	bSetParameter					: BOOL;
	bConnect						: BOOL := TRUE;
	bIncommingMsg					: BOOL;
	hrErrorOccurred 				: DINT; //Contains latest error message
	sTopicRec						: STRING(255);
	sMessage						: STRING(255);
	ReinitComParams					: BOOL;
	
	
	bSubscribed						: BOOL;
	ton_PublishInterval				: TON;
	sPubTopic						: STRING;
	sSubTopic						: STRING;
	
	stPubDataMaster					: ST_InterMachineCom_Master;
	stPubDataSlave					: st_InterMachineCom_Slave;
	stSubDataMaster					: ST_InterMachineCom_Master;
	stSubDataSlave					: st_InterMachineCom_Slave;
	
	
	fbJson         	: FB_JsonSaxWriter;
  	fbJsonDataType 	: FB_JsonReadWriteDataType;
	sJsonDocPub     : STRING(255);
	bRecJsonOK		: BOOL;
	
	
	sMasterTopic 	: STRING := 'master';
END_VAR

(* 
Internal broker is used to post local data in the master topic. The unit listens to the slave topics

*)

//Connect brokers

//Generate machinedata for internal master
InternalBroker(bConnect := TRUE, sHostname := ST_params.InternalBrokerIP);
InternalBroker.Publish(
	Interval := st_params.MasterPublishRate, 
	sTopic := sMasterTopic, 
	sMessage := StructToJson(TRUE));
InternalBroker.Subscribe(sTopic := 'slave/epu/#/read');

IF internalbroker.bIncomingMsg THEN
	JsonToStruct(sMessage := internalbroker.sMessage);
END_IF

//Generate slave data for the external master
ExternalBroker(bConnect := SlaveConnectionData.enable, sHostname := SlaveConnectionData.BrokerIP);
ExternalBroker.Publish(Interval := st_params.SlavePublishRate, 
		sTopic := CONCAT(CONCAT('epu/slave/',settings.Properties.s_SerialNumber),'/read'),
		sMessage := StructToJson(FALSE));
ExternalBroker.Subscribe(sTopic := sMasterTopic);

IF Externalbroker.bIncomingMsg THEN
	JsonToStruct();
END_IF




//Publish as master 
sPubTopic := 'master';
sSubTopic := 'slave/#';
//Ton_PublishInterval.PT := st_params.MasterPublishRate;
//generate json doc
fbJson.ResetDocument();
fbJsonDataType.AddJsonValueFromSymbol(fbJson, 'ST_InterMachineCom_Master', SIZEOF(stPubDataMaster), ADR(stPubDataMaster));
fbJson.EndObject();
fbJson.CopyDocument(sJsonDocPub, SIZEOF(sJsonDocPub));

IF SlaveConnectionData.enable AND SlaveConnectionData.BrokerIP <> '' THEN
	sSubTopic := 'master';
	sPubTopic := CONCAT('slave/', settings.Properties.s_SerialNumber);
	Ton_PublishInterval.PT := st_params.MasterPublishRate;
	//generate json doc
	fbJson.ResetDocument();
	fbJsonDataType.AddJsonValueFromSymbol(fbJson, 'ST_InterMachineCom_Slave', SIZEOF(stPubDataSlave), ADR(stPubDataSlave));
	fbJson.EndObject();
	fbJson.CopyDocument(sJsonDocPub, SIZEOF(sJsonDocPub));
	
	//converter receiving message back to structur
	fbJsonDataType.SetSymbolFromJson(sMessage, 'st_InterMachineCom_Master', SIZEOF(stSubDataMaster), ADR(stSubDataMaster));
END_IF

// publish
IF fbMqttClientInternal.bConnected THEN
    IF NOT bSubscribed THEN
        bSubscribed := fbMqttClientInternal.Subscribe(sTopic:=sSubTopic, eQoS:=TcIotMqttQos.AtMostOnceDelivery); //sSubTopic
    END_IF
    ton_PublishInterval(IN:=TRUE);
    IF ton_PublishInterval.Q THEN // publish new payload every second
        ton_PublishInterval(IN:=FALSE);
			fbMqttClientInternal.Publish(sTopic:=sPubTopic,
			pPayload := ADR(sJsonDocPub),
			nPayloadSize := LEN2(ADR(sJsonDocPub)),
			eQoS := TcIotMqttQos.AtMostOnceDelivery,
			bRetain:= TRUE,
			bQueue := FALSE);
    END_IF
END_IF


IF bIncommingMsg THEN
	bRecJsonOK := fbJsonDataType.SetSymbolFromJson(sMessage, 'st_InterMachineCom_Slave', SIZEOF(stSubDataSlave), ADR(stSubDataSlave));
END_IF

Internalbroker.Subscribe();

METHOD CheckSlaves : BOOL
VAR_INPUT
END_VAR
END_METHOD

METHOD GetSubData : BOOL
VAR_INPUT
END_VAR
END_METHOD

METHOD JsonToStruct : BOOL
VAR_INPUT
	MasterMode		: BOOL;
END_VAR

VAR_IN_OUT
	sMessage : STRING;
END_VAR
IF MasterMode THEN
	//Get the message from the external broker 'master' subscribtion, format according to ST_IntermachineCom_Master
ELSE
	//Get the message from the internal broker '+/slave/#/read' subscriptiom, format according to ST_intermachineCom_Slave
	(* A json parser need to be constructed such that the combined json struct is formatted in separate st_IntermachineCom_slave structs.
	
	Data can come from the epu or hpu and distinquish is made through the topic path: /slave/hpu/#, or /slave/epu/#
	For example the epu slave path is: /slave/epu/{serialnumber}/read and the ST_intermachineCom_slave struct comes out.
	A json filter has to be made to iterate along all serial numbers in epu and hpu group. 
	A method must be created where the data is temporarily stored such that the ACP (available charge power), 
	ADP (available discharge power) and ARP (available reactive power) can me summed and used for the power setpoint calculation.
	
	A separate topic /slave/epu/{serialnumber}/write can be used to control slaves individually with the ST_IntermachineCom_master struct.
	However, this requires the slave CW heartbeat and SW heartbeat to be updated within heartbeat time limit. When the CW heartbeat stops, 
	the slave will go to general operation related to the 'master' topic that is broadcasted. 
	*)
END_IF
END_METHOD

METHOD Reset : BOOL
VAR_INPUT
END_VAR
IF InternalBroker.bRestartConnection AND ExternalBroker.bRestartConnection THEN
	InternalBroker.bRestartConnection := FALSE;
	ExternalBroker.bRestartConnection := FALSE;
	Reset := TRUE;
ELSE
	InternalBroker.bRestartConnection := NOT InternalBroker.bRestartConnection;
	ExternalBroker.bRestartConnection := NOT ExternalBroker.bRestartConnection;
END_IF
END_METHOD

METHOD SetPubData : BOOL
VAR_INPUT
END_VAR

VAR_INST
	WatchdogPulse	: TON; 
END_VAR
WatchdogPulse(IN := NOT watchdogPulse.Q, PT:= st_params.WatchdogPulseRate);

//Internal 'master' data to control slaves
stPubDataMaster.CW.0 := monitor.powerstack.b_StartedState;
stPubDataMaster.CW.1 := monitor.powerstack.e_State = eStatusPowerstack.idle;
stPubDataMaster.CW.2 := monitor.powerstack.e_State = eStatusPowerstack.shutdown;
stPubDataMaster.CW.3 := GVL.b_EmergencyShutdownActive AND ST_IntermachineCom_params.EMstopCoupling;
stPubDataMaster.CW.4 := monitor.system.e_State = eSystemState.Reset;
stPubDataMaster.CW.15 := SEL(watchdogPulse.Q, stPubDataMaster.CW.15, NOT stPubDataMaster.CW.15);
stPubDataMaster.PS := 0; // TBD based on slaves
stPubDataMaster.QS := 0; 

//Slave data for external master
stPubDataSlave.ACP := TO_UINT(ABS(monitor.powerstack.r_Pmin));
stPubDataSlave.ADP := TO_UINT(ABS(monitor.powerstack.r_PMax));
stPubDataSlave.AQ := TO_UINT(ABS(monitor.powerstack.r_QMax));
stPubDataSlave.SW.0 := monitor.system.e_State = eSystemState.StandBy OR monitor.system.e_State = eSystemState.Conditioning;
stPubDataSlave.SW.1 := monitor.powerstack.b_StartedState;
stPubDataSlave.SW.2 := monitor.system.e_State = eSystemState.Stopped;
stPubDataSlave.SW.3 := monitor.system.e_State = eSystemState.Discharging_Only;
stPubDataSlave.SW.4 := monitor.system.e_State = eSystemState.Charging_Only;
stPubDataSlave.SW.5 := GVL.b_WarningActive;
stPubDataSlave.SW.6 := GVL.b_NormalShutdownActive;
stPubDataSlave.SW.7 := GVL.b_EmergencyShutdownActive;
stPubDataSlave.SW.15 := stSubDataMaster.CW.15;
END_METHOD

METHOD StructToJson : STRING
VAR_INPUT
	Mastermode		: BOOL; //if false, then slave mode
END_VAR
fbJson.ResetDocument();

IF MasterMode THEN
	fbJsonDataType.AddJsonValueFromSymbol(fbJson, 'ST_InterMachineCom_Master', SIZEOF(stPubDataMaster), ADR(stPubDataMaster));
ELSE
	fbJsonDataType.AddJsonValueFromSymbol(fbJson, 'ST_InterMachineCom_Slave', SIZEOF(stPubDataSlave), ADR(stPubDataSlave));
END_IF

fbJson.EndObject();
fbJson.CopyDocument(StructToJson, SIZEOF(StructToJson));
END_METHOD

END_FUNCTION_BLOCK

// ---- POUs/Objects/PLCStatus/FB_PLCUpdate.TcPOU
FUNCTION_BLOCK FB_PLCUpdate

VAR_INPUT
	bUpdate				: BOOL;
	bAbortUpdate		: BOOL;
END_VAR

VAR_OUTPUT
	FTPState			: eFTPstate;
	InstalState			: eInstalState;
	BackupState			: eInstalState;
	sLogMessage 		: STRING(255);
	bCheckUpdates		: BOOL;	
	bUpdateAvailable 	: BOOL;
END_VAR

VAR	
	rTrig_CheckUpdate	: R_Trig;
	
    fbFileDelete 		: FB_FileDelete;  (* Om oude bestanden te verwijderen *)
    
    sJsonUrl      		: STRING := 'http://server.com/updates.json'; (* JSON met update-info *)
    sUpdateUrl    		: STRING := '';  (* URL van het updatebestand uit JSON *)
    sLocalPath    		: STRING := '/usr/local/updates/update.tsmpkg';
    sBackupPath   		: STRING := '/usr/local/backup/old_version.tsmpkg';
    
    sCurrentVersion 	: STRING := '1.2.0';  (* Huidige versie van de PLC *)
    sNewVersion     	: STRING := '';       (* Nieuwe versie uit JSON *)

   
    bDownloadComplete 	: BOOL;
    bInstallComplete 	: BOOL;
    bRollbackNeeded 	: BOOL;
    eState 				: INT := 0;
    iRetryCount 		: INT := 0;
END_VAR




CASE eState OF
    0: // Controleer op update via JSON
		rTrig_CheckUpdate(CLK := bUpdate);
		IF rTrig_CheckUpdate THEN
			bCheckUpdates := TRUE;
		END_IF
		
		IF 
		CheckForUpdates();
        

    1: // Maak een backup van de huidige versie
		BackupState := Copy(sSrcPath := sLocalPath, sDestPath := sBackupPath);
		
        IF BackupState = eInstalState.Success THEN
            eState := 2;
		ELSIF BackupState = eInstalState.Failure OR bAbortUpdate THEN
			eState := 99;
        END_IF

    2: // Download de nieuwe update via FTP
		FTPState := DownloadUpdate(
			sHost := 'temp',
			sUsername := 'tempuser',
			sPassword := 'tempPass',
			sSrcFile := 'path/1',
			sDesFile := 'path/2',
			start :=  bUpdateAvailable);

        IF FTPState = eFTPState.Success THEN
            bDownloadComplete := TRUE;
            eState := 3;
        ELSIF FTPState = eFTPState.Failure OR bAbortUpdate THEN
                eState := 99; // Ga naar fallback
        END_IF

    3: // Wachten op bevestiging van de gebruiker via HMI
        IF bUpdate THEN
			bUpdateStarted := TRUE;
            eState := 4;
        END_IF

    4: // Installeer de update
		InstalState := Copy(sSrcPath := sLocalPath, sDestPath := 'path/2');
		IF InstalState = eInstalState.Success THEN
			bInstallComplete := TRUE;
			eState := 5;
		ELSIF InstalState = eInstalState.Failure OR bAbortUpdate THEN
			bRollbackNeeded := TRUE;
            eState := 6; // Ga naar rollback
		END_IF

    5: // Herstart de PLC na succesvolle update
        SystemReboot();

    6: // Rollback uitvoeren als de update is mislukt
		InstalState := Copy(sSrcPath := sBackupPath,  sDestPath := '/usr/local/boot/update.tsmpkg');

		IF InstalState = eInstalState.Success THEN
			SystemReboot();  // Herstart de PLC met oude versie
		ELSIF InstalState = eInstalState.Failure OR bAbortUpdate THEN
			eState := 99;  // Fallback activeren als rollback mislukt
		END_IF

    99: // Fallback: Stop het updateproces en meld de fout
        bUpdateAvailable := FALSE;
		bUpdateStarted := FALSE;
        bRollbackNeeded := FALSE;
        iRetryCount := 0;
END_CASE

CASE eState OF
    0:	sLogMessage := 'Check if update is available';
        WriteLog(sLogMessage);
        
   1:	sLogMessage := 'Create backup of current software';
        WriteLog(sLogMessage);

    2:	sLogMessage := 'Downloading update';
        WriteLog(sLogMessage);
		
	3:	sLogMessage := 'Update ready for installation';
		WriteLog(sLogMessage);
		
	4:	sLogMessage := 'Installing update';
		WriteLog(sLogMessage);
		
	5:	sLogMessage := 'Rebooting system';
		WriteLog(sLogMessage);    
		
    6:	sLogMessage := 'Update failed, rollback started';
         WriteLog(sLogMessage);
		 
    99:
        sLogMessage := 'Update mislukt, fallback geactiveerd';
        WriteLog(sLogMessage);
END_CASE

METHOD CheckForUpdates : BOOL
VAR_INPUT
	sServerUrl   : STRING := 'http://server.com/updates.json'; (* Volledige URL *)
END_VAR

VAR_INST
	fbHttpClient 		: FB_IotHttpClient;  (* Voor JSON versiecontrole *)
	     
    sResponse    : STRING(1024);  (* Buffer voor de server response *)
    bExecute     : BOOL := TRUE;
    bDone        : BOOL;
    bError       : BOOL;
END_VAR
fbHttpClient(
	sHostName := sHostName,
	


fbHttpClient.sHost := 'server.com';  // Vervang met je eigen server
fbHttpClient.sResource := '/updates.json';  // JSON-bestand
fbHttpClient.eMethod := E_HttpMethod.GET;
fbHttpClient.bExecute := TRUE;

IF fbHttpClient.eState = E_HttpRequestState.Done THEN
	sNewVersion := ExtractJsonValue(fbHttpClient.sResponseContent, 'latest_version');
	sUpdateUrl := ExtractJsonValue(fbHttpClient.sResponseContent, 'update_file');
	
	IF sNewVersion > sCurrentVersion THEN
		bUpdateAvailable := TRUE;
		eState := 1;
	END_IF
END_IF


(* Stap 1: HTTP Request starten *)
IF bExecute THEN
    fbHttpClient. := sServerUrl;   (* Geef de volledige URL mee *)
    fbHttpClient.eMethod := T_IotHttpMethod.Get;  (* HTTP GET Methode *)
    fbHttpClient.bExecute := TRUE;
    bExecute := FALSE; (* Voorkomt dat het telkens opnieuw start *)
END_IF

(* Stap 2: Wachten op antwoord *)
IF fbHttpClient.bDone THEN
    sResponse := fbHttpClient.sResponse;  (* Server response opslaan *)
    bDone := TRUE;
ELSIF fbHttpClient.bError THEN
    bError := TRUE;
END_IF
END_METHOD

METHOD Copy : eInstalstate
VAR_INPUT
	sSrcPath : STRING;
	sDestPath: STRING;
END_VAR

VAR_OUTPUT
	Busy 		: BOOL;
    Error 		: BOOL;
	ErrID 		: UDINT;
END_VAR

VAR_INST
	ton_waitRetry		: ton := (pt := T#2S);
	fbFileCopy   		: FB_FileCopy;    (* Voor het maken van een backup *)
END_VAR
fbFileCopy(
	sSrcPathName := sSrcPath,
	sDestPathName := sDestPath,
	tTimeOut := T#15S,
	bBusy => Busy,
	bError => Error,
	nErrId => ErrID);
	
ton_waitRetry(Q => fbFileCopy.bExecute);

IF Error THEN
	Copy := eInstalState.Failure;
ELSIF busy THEN
	Copy := eInstalState.InProgress;
	ton_waitRetry.IN := FALSE;
ELSE
	IF NOT fbFileCopy.bExecute THEN
		Copy := eInstalState.Success;
	END_IF
	ton_waitRetry.IN := TRUE;
END_IF
END_METHOD

METHOD DownloadUpdate : eFTPState

VAR_INPUT
	sHost 			: STRING := 'ftp.example.com';
	sUsername		: STRING;
	sSrcFile		: STRING;
	sDesFile		: STRING;
	sPassword		: STRING;
	Start			: BOOL;
END_VAR

VAR_OUTPUT
	Busy 		: BOOL;
    Error 		: BOOL;
	ErrID 		: UDINT;
END_VAR

VAR_INST
	bRetry			: BOOL;
	byMaxRetries	: BYTE := 3;
	byRetryCounter	: BYTE;
	StartTrigger : R_TRIG;	
	FTPstate 	: eFTPState;
	ftpOpen 	: FB_FTP_Open; 			// Function block om verbinding te openen.
	ftpDownload : FB_FTP_FileDownload; 	// Function block om het bestand te downloaden
    ftpClose 	: FB_FTP_Close;  			// Function block om de verbinding te sluiten
    hFTP 		: T_HFTP; //FTP handle / identifyer
	RTrig_Error	: R_Trig;
END_VAR
StartTrigger(CLK:= start);

CASE FTPState OF
      eFTPState.Disconnected:
			IF StartTrigger.Q OR bRetry THEN
				bRetry := FALSE;
      			FTPState := eFTPState.Connecting;
			END_IF
			
     eFTPState.Connecting:
         ftpOpen(
			sHost:= sHost,
			nPort:= 21,
			sUsername:= sUsername,
			sPassword:= sPassword,
			tTimeout:= T#15S,
			bExecute := TRUE,
			hFTP=> hFTP,
			bBusy => busy,
			bError => Error,
			nErrID=> ErrID
			);
         IF NOT Busy AND NOT Error THEN
             ftpOpen(bExecute:= FALSE);
             FTPState := eFTPstate.Downloading;
         END_IF
		 
     eFTPstate.Downloading:
		ftpDownload(
			sNetID:= '',              // Lokale machine
			hFTP:= hFTP,              // Gebruik de handle van de geopende verbinding
			sSrcFile:= '\TestFolder\File1.txt',
            sDesFile:= '\Program Files\TestFile1.txt',
			tTimeout:= T#15S,         // Timeout
			bexecute := TRUE,
			bBusy => busy,
            bError => error,
			nErrID=> ErrID
		);
         IF NOT busy AND NOT Error THEN
             ftpDownload(bExecute:= FALSE);
             FTPState := eFTPState.Success;
         END_IF
     eFTPState.Success:
		ftpClose(
			sNetID:= '',              // Lokale machine
			hFTP:= hFTP,              // Gebruik de handle van de geopende verbinding
			bExecute:= TRUE,      // Start het sluiten van de verbinding
			bBusy => busy,
            bError => error,
			tTimeout:= T#15S,         // Timeout
			nErrID=> ErrID
		);
	 	
       	 IF NOT busy AND NOT Error THEN
             ftpClose(bExecute:= FALSE);
             FTPstate := eFTPState.Disconnected;
			 byRetryCounter := 0;
         END_IF
		
	eFTPState.Failure:
		IF StartTrigger.Q THEN
			FTPState := eFTPState.Connecting;
		END_IF	 	
END_CASE

//Retry on error trigger
RTrig_Error(CLK:= Error);
IF RTrig_Error.Q THEN
	IF ByRetryCounter < byMaxRetries THEN
		FTPstate := eFTPState.Disconnected;
		bRetry := TRUE;
		byRetryCounter := byRetryCounter +1;
	ELSE
		FTPstate := eFTPState.Failure;
	END_IF
END_IF

DownloadUpdate := FTPState;
END_METHOD

METHOD SystemReboot : BOOL
VAR_INPUT
END_VAR

VAR_INST
    fbSysRestart 		: TC_Restart; (* Systeemherstartfunctie *)
END_VAR
fbSysRestart();
END_METHOD

METHOD WriteLog : BOOL
VAR_INPUT
    sMessage : STRING;
END_VAR

VAR_INST
    fbLogWriter 		: FB_FileWrite;
END_VAR
fbLogWriter(
fbLogWriter.sFileName := '/usr/local/logs/update_log.txt';
fbLogWriter.sData := sMessage + Char(13) + Char(10);
fbLogWriter.bExecute := TRUE;
WriteLog := fbLogWriter.bDone;
END_METHOD

END_FUNCTION_BLOCK

// ---- POUs/System/PowerControl/fb_measurementCheck.TcPOU
FUNCTION_BLOCK fb_measurementCheck
VAR_IN_OUT
	r_in : REAL;
END_VAR
VAR_INPUT
	b_externalFault : BOOL;
	r_LowLimit	 	: REAL;
	r_HighLimit		: REAL;
	by_Mode			: BYTE := 0; // 0= min, 1= avg, 2= Max, 3=SUM
END_VAR

VAR
	by_InputOK		: BYTE;
END_VAR

VAR_OUTPUT
	r_Out			: REAL;
	Q				: BOOL;
END_VAR


//Check if values are within set ranges
by_InputOK.0 := r_in > r_LowLimit AND r_in < r_HighLimit;
by_InputOK.1 := r_in[Phases.L1] > r_LowLimit AND r_in[phases.L1] < r_HighLimit;
by_InputOK.2 := r_in[Phases.L2] > r_LowLimit AND r_in[phases.L2] < r_HighLimit;
by_InputOK.3 := r_in[Phases.L3] > r_LowLimit AND r_in[phases.L3] < r_HighLimit;

//Check if deviation between values is not too high

IF by_InputOK >= 14 AND NOT b_ExternalFault THEN // 14 == L1, L2, L3 OK
	CASE by_Mode OF
		0: r_out := MIN(r_in[1], r_in[2], r_in[3]); //MIN
		1: r_out := (r_in[1] + r_in[2] + r_in[3]) / 3; // AVG
		2: r_out := MAX(r_in[1], r_in[2], r_in[3]); //MAX
		3: r_out := r_in[1] + r_in[2] + r_in[3]; //sum
		4: r_out := MAX(ABS(r_in[1]), ABS(r_in[2]), ABS(r_in[3])) * 3 * SEL(r_in[1] + r_in[2] + r_in[3] < 0, 1, -1); //sum
	END_CASE
	Q := TRUE;
ELSIF by_InputOK = 1 THEN
	r_Out := r_in[0];
ELSE
	r_out := 0;
	Q := FALSE;
END_IF

END_FUNCTION_BLOCK
